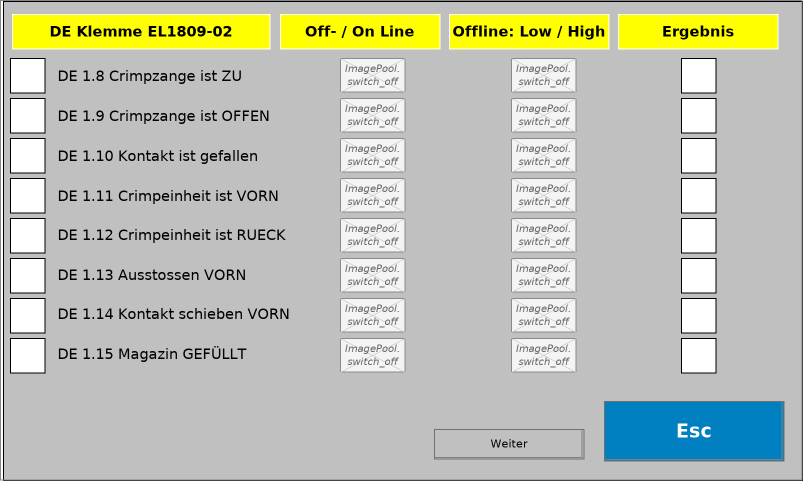
VISUALIZATION IO_Visu02  // 803x481
    Rectangle (3,1 800x480)
    Label (50,61 271x30), "DE 1.8 Crimpzange ist ZU"
    Rectangle (12,14 258x35), "DE Klemme EL1809-02"
    Label (50,101 279x30), "DE 1.9 Crimpzange ist OFFEN"
    Label (50,141 269x30), "DE 1.10 Kontakt ist gefallen"
    Label (50,181 277x30), "DE 1.11 Crimpeinheit ist VORN"
    Label (50,220 283x30), "DE 1.12 Crimpeinheit ist RUECK"
    Label (50,260 278x30), "DE 1.13 Ausstossen VORN"
    Label (50,299 292x30), "DE 1.14 Kontakt schieben VORN"
    Rectangle (10,58 35x35), colour toggle: IO.inCrimpZangeIstZU
    Rectangle (10,98 35x35), colour toggle: IO.inCrimpZangeIstOFFEN
    Rectangle (10,138 35x35), colour toggle: IO.inKontaktIstGefallen
    Rectangle (10,178 35x35), colour toggle: IO.inCrimpEinheitIstVORN
    Rectangle (10,218 35x35), colour toggle: IO.inCrimpEinheitIstRUECK
    Rectangle (10,258 35x35), colour toggle: IO.inAusstossenVORN
    Rectangle (10,298 35x35), colour toggle: IO.inKontaktSchiebenVORN
    Rectangle (10,338 35x35), colour toggle: IO.inMagazinGEFUELLT
    Label (50,339 300x30), "DE 1.15 Magazin GEFÜLLT"
    Rectangle (280,14 160x35), "Off- / On Line"
    Image (340,58 65x34), image: ImagePool.switch_off
        p84334746: P_InputHandling.E1_8.onlineImageID
        OnMouseUp: execute { RVL.e18Online := NOT RVL.e18Online; }
    Image (340,98 65x34), image: ImagePool.switch_off
        p84334746: P_InputHandling.E1_9.onlineImageID
        OnMouseUp: execute { RVL.e19Online := NOT RVL.e19Online; }
    Image (340,138 65x34), image: ImagePool.switch_off
        p84334746: P_InputHandling.E1_10.onlineImageID
        OnMouseUp: execute { RVL.e110Online := NOT RVL.e110Online; }
    Image (340,178 65x34), image: ImagePool.switch_off
        p84334746: P_InputHandling.E1_11.onlineImageID
        OnMouseUp: execute { RVL.e111Online := NOT RVL.e111Online; }
    Image (340,218 65x34), image: ImagePool.switch_off
        p84334746: P_InputHandling.E1_12.onlineImageID
        OnMouseUp: execute { RVL.e112Online := NOT RVL.e112Online; }
    Image (340,258 65x34), image: ImagePool.switch_off
        p84334746: P_InputHandling.E1_13.onlineImageID
        OnMouseUp: execute { RVL.e113Online := NOT RVL.e113Online; }
    Image (340,298 65x34), image: ImagePool.switch_off
        p84334746: P_InputHandling.E1_14.onlineImageID
        OnMouseUp: execute { RVL.e114Online := NOT RVL.e114Online; }
    Image (340,338 65x34), image: ImagePool.switch_off
        p84334746: P_InputHandling.E1_15.onlineImageID
        OnMouseUp: execute { RVL.e115Online := NOT RVL.e115Online; }
    Rectangle (449,14 160x35), "Offline: Low / High"
    Image (511,58 65x34), image: ImagePool.switch_off
        p84334746: P_InputHandling.E1_8.modeImageID
        OnMouseUp: execute { RVL.e18OffMode := NOT RVL.e18OffMode; }
    Image (511,98 65x34), image: ImagePool.switch_off
        p84334746: P_InputHandling.E1_9.modeImageID
        OnMouseUp: execute { RVL.e19OffMode := NOT RVL.e19OffMode; }
    Image (511,138 65x34), image: ImagePool.switch_off
        p84334746: P_InputHandling.E1_10.modeImageID
        OnMouseUp: execute { RVL.e110OffMode := NOT RVL.e110OffMode; }
    Image (511,178 65x34), image: ImagePool.switch_off
        p84334746: P_InputHandling.E1_11.modeImageID
        OnMouseUp: execute { RVL.e111OffMode := NOT RVL.e111OffMode; }
    Image (511,218 65x34), image: ImagePool.switch_off
        p84334746: P_InputHandling.E1_12.modeImageID
        OnMouseUp: execute { RVL.e112OffMode := NOT RVL.e112OffMode; }
    Image (511,258 65x34), image: ImagePool.switch_off
        p84334746: P_InputHandling.E1_13.modeImageID
        OnMouseUp: execute { RVL.e113OffMode := NOT RVL.e113OffMode; }
    Image (511,298 65x34), image: ImagePool.switch_off
        p84334746: P_InputHandling.E1_14.modeImageID
        OnMouseUp: execute { RVL.e114OffMode := NOT RVL.e114OffMode; }
    Image (511,338 65x34), colour toggle: GVL.insecAbisoliererIstLINKS, image: ImagePool.switch_off
        p84334746: P_InputHandling.E1_15.modeImageID
        OnMouseUp: execute { RVL.e115OffMode := NOT RVL.e115OffMode; }
    Rectangle (681,58 35x35), colour toggle: GVL.insecCrimpZangeIstZU
    Rectangle (681,98 35x35), colour toggle: GVL.insecCrimpZangeIstOFFEN
    Rectangle (681,138 35x35), colour toggle: GVL.insecKontaktIstGefallen
    Rectangle (681,178 35x35), colour toggle: GVL.insecCrimpEinheitIstVORN
    Rectangle (681,218 35x35), colour toggle: GVL.insecCrimpEinheitIstRUECK
    Rectangle (681,258 35x35), colour toggle: GVL.insecAusstossenVORN
    Rectangle (681,298 35x35), colour toggle: GVL.insecKontaktSchiebenVORN
    Rectangle (681,338 35x35), colour toggle: GVL.insecMagazinGEFUELLT
    Rectangle (618,14 160x35), "Ergebnis"
    Button (434,429 150x30), "Weiter"
        OnMouseClick: change screen: IO_Visu01
    Button (604,401 180x60), "Esc"
        OnMouseUp: change screen: Menu
END_VISUALIZATION

(* stored: Version 1.1.0.1, ProductVersion 3.1.4024.3
   Visu IO_Visu02: Id {34ff36c1-8530-4389-b99f-aaad0b1f0819} *)
